PROGRAM MAIN
VAR
	fbController		:	FB_Controller();
	eActiveLamp 		:	E_LampType;
	bSetActiveLamp 		:	BOOL;
	bDimUp, bDimDown	:	BOOL;
	bOff, bOn			:	BOOL;
END_VAR

IF (bSetActiveLamp) THEN
	fbController.eActiveLamp := eActiveLamp;
	bSetActiveLamp := FALSE;
END_IF

IF (bDimUp) THEN
	fbController.DimUp();
	bDimUp := FALSE;
END_IF

IF (bDimDown) THEN
	fbController.DimDown();
	bDimDown := FALSE;
END_IF

IF (bOff) THEN
	fbController.Off();
	bOff := FALSE;
END_IF

IF (bOn) THEN
	fbController.On();
	bOn := FALSE;
END_IF

END_PROGRAM

(* stored: Version 1.1.0.1, ProductVersion 3.1.4024.6
   POU MAIN: Id {ef33b4c1-c95d-4cf8-b9bf-7d346bd93484}, SpecialFunc None *)
